// TIA Portal V19 export
FUNCTION_BLOCK "UP_Spuele.GP0x"   // FB1003, LAD
TITLE = Umwälzpumpe Spüle
{ S7_Optimized_Access := 'TRUE' }
// Funktionen:  Entleeren /  Spülen
// stored: AutoNumber false, MemoryReserve 100, SetENOAutomatically false
   VAR RETAIN
      In { ExternalAccessible := 'False'; ExternalVisible := 'False'; ExternalWritable := 'False'} : Struct
         NotHalt : Bool;
         ext_Freigabe : Bool;   // kein Gasalarm, Kein Notstrom
         TW_senkt : Bool;
         Auto : Bool;   // Paneltaste
         Ein : Bool;   // Paneltaste
         FU_betriebsbereit : Bool;
         FU_Stoerung : Bool;
         Niv_TLS : Bool;
         Niv_min : Bool;
         Frg_Niv_CM05 : Bool;
         SRM_Saugseite_auf : Bool;
         SRM_Saugseite_zu : Bool;
         SRM_Druckseite_auf : Bool;
         SRM_Druckseite_zu : Bool;
         GW_p_UP : Bool;
         Betriebsart : USInt := 0;   // Paneltaste
         FU_speed : Int;
         Druck_Pumpe : Real;
      END_STRUCT;
      Param { ExternalAccessible := 'False'; ExternalVisible := 'False'; ExternalWritable := 'False'} : Struct
         SW_Hand : Int;   // [%]
         SW_Auto_AZ : Int;   // [%]
         SW_Auto_aAZ : Int;   // [%]
         Spülzeit : Time;
         DT_Druckaufbau : Time;
         DT_Testzeit : Time;
         SW_Drucktest : Real;
         "Name" : String[12];
      END_STRUCT;
      Zst { ExternalAccessible := 'False'; ExternalVisible := 'False'; ExternalWritable := 'False'} : Struct
         Niveau : USInt;
         Status_GP0x : USInt;
         Status_DT : USInt;
         Restzeit_Spülen : Time;
         Restzeit_DT : Time;
         TON_Spülventil_auf : Bool;
         Spuelen : Bool;
         Spuelen_aktiv : Bool;
         Drucktest_aktiv : Bool;
         Umwaelzen : Bool;
         Zeit_laeuft : Bool;
         Drucktest_ok : Bool;
         Bedienung_erlaubt : Bool;
         speed : Int;   // [%]
      END_STRUCT;
      Mld { ExternalAccessible := 'False'; ExternalVisible := 'False'; ExternalWritable := 'False'} : Struct
         Niv_TLS : Bool;
         Niv_Sensorfehler : Bool;
         GW_p_UP : Bool;
         FU_nicht_bereit : Bool;
         FU_Stoerung : Bool;
         n_Auto : Bool;
         TO_Druckaufbau : Bool;
         Drucktest_ok : Bool;
         DT_Fehler : Bool;
         Pu_Spuelen_Fertig : Bool;
      END_STRUCT;
      Out { ExternalAccessible := 'False'; ExternalVisible := 'False'; ExternalWritable := 'False'} : Struct
         GP0x_Ein : Bool;
         Ventil_Saugseite : Bool;
         Ventil_Druckseite : Bool;
         Spülventil : Bool;
         Ventil_CM05 : Bool;
         Soll_speed : Int;
      END_STRUCT;
   END_VAR
   VAR
      IEC_Timer { ExternalAccessible := 'False'; ExternalVisible := 'False'; ExternalWritable := 'False'} : Struct
         Spülventil_auf { S7_SetPoint := 'True'} : TON_TIME;
         Spülen { S7_SetPoint := 'True'} : TP_TIME;
         GW_p { S7_SetPoint := 'True'} : TON_TIME;
         Drucktest { S7_SetPoint := 'True'} : TP_TIME;
         TO_Druckaufbau { S7_SetPoint := 'True'} : TON_TIME;
         Ventil_CMO5 { S7_SetPoint := 'True'} : TOF_TIME;
      END_STRUCT;
      R_TRIG_Hand_EIN { ExternalAccessible := 'False'; ExternalVisible := 'False'; ExternalWritable := 'False'} : R_TRIG;
   END_VAR
   VAR_TEMP
      Spülzeit : Time;
      Zeit_DT : Time;
      posFl_Hand : Bool;
   END_VAR
   VAR CONSTANT
      Niv_TLS : USInt := 7;
      Niv_Min : USInt := 70;
      Niv_max : USInt := 85;
      Zeit_Ventil_auf : Time := T#1s;
      S1 : USInt := 1;
      S2 : USInt := 2;
      S3 : USInt := 3;
      S4 : USInt := 4;
   END_VAR
BEGIN

REGION Network 1 (SCL): Input
   // Panelbedienung und Sensoren --> Input()
   // Not-Halt
   #In.NotHalt := NOT "DB_PNOZ_IN_Out".In.NH_Frg_Pumpen OR NOT "E_Frg_AbLW";

   // Timer Spülventil AUF
   #IEC_Timer.Spülventil_auf(IN := #Out.Spülventil,
                              PT := #Zeit_Ventil_auf,
                              Q => #Zst.TON_Spülventil_auf);

    // positive Flanke "Hand Ein"
   #R_TRIG_Hand_EIN(CLK := #In.Ein,
                    Q => #posFl_Hand);
END_REGION

REGION Network 2 (SCL): Ansteuerung

   // "Normal"-Betrieb
   #Zst.Bedienung_erlaubt := NOT #In.Ein AND NOT #In.Auto AND NOT #Mld.DT_Fehler;

   //Drucktest rücksetzen
   IF #In.Betriebsart <> 2 OR #Zst.Spuelen_aktiv OR #Zst.Umwaelzen OR NOT #In.Ein THEN
       #Mld.Drucktest_ok := FALSE;
       // #Mld.DT_Fehler := FALSE;
       #Mld.TO_Druckaufbau := FALSE;
       #Zst.Status_DT := 0;
       #Zst.Drucktest_aktiv := FALSE;
   END_IF;
   //Spülmeldung rücksetzen
   IF #In.Betriebsart <> 1 OR NOT #In.Ein THEN
       #Mld.Pu_Spuelen_Fertig := FALSE;
   END_IF;

       CASE #In.Betriebsart OF
           0:  // Umwälzen

               // Spülventil zu
               #Out.Spülventil := FALSE;
               #Out.Ventil_CM05 := FALSE;
               #Zst.Restzeit_Spülen := T#0s;
               // Ventile öffnen
               #Out.Ventil_Saugseite := (#In.Auto OR #In.Ein) AND #In.Niv_TLS AND NOT #In.TW_senkt;
               #Out.Ventil_Druckseite := #Out.Ventil_Saugseite;
               // Wenn geöffnet --> Frg Pumpe
               #Zst.Umwaelzen := #In.SRM_Druckseite_auf AND #In.SRM_Saugseite_auf;
               #Zst.Drucktest_aktiv := FALSE;

           1: // Spülen - nur Hand
               #Zst.Umwaelzen := FALSE;
               #Out.Ventil_Saugseite := FALSE;
               #Out.Ventil_Druckseite := FALSE;

               // Ausschaltverzögert - Druckabbau
               #IEC_Timer.Ventil_CMO5(IN := #Out.Spülventil,
                                      PT := T#3s,
                                      Q => #Out.Ventil_CM05);

                   IF #In.Ein AND #In.Frg_Niv_CM05 THEN
                       IF #posFl_Hand THEN
                           #Zst.Spuelen_aktiv := TRUE;
                       END_IF;

                       #Out.Spülventil := #In.SRM_Druckseite_zu AND #In.SRM_Saugseite_zu AND #Zst.Spuelen_aktiv;

                       #IEC_Timer.Spülen(IN := #Zst.TON_Spülventil_auf,
                                         PT := #Param.Spülzeit,
                                         Q => #Zst.Spuelen,
                                         ET => #Spülzeit);
                       #Zst.Restzeit_Spülen := #Param.Spülzeit - #Spülzeit;

                       IF #Zst.TON_Spülventil_auf AND #In.SRM_Saugseite_zu AND #In.SRM_Druckseite_zu
                           AND NOT #Zst.Spuelen AND #Zst.Spuelen_aktiv THEN
                           #Zst.Spuelen_aktiv := FALSE;
                           #Out.Spülventil := FALSE;
                       END_IF;

                       // Fertig
                       IF NOT #Zst.Spuelen AND NOT #Zst.Spuelen_aktiv AND NOT #Out.Ventil_CM05 THEN
                           #Out.Spülventil := FALSE;
                           #Out.Ventil_CM05 := FALSE;
                           #Zst.Restzeit_Spülen := T#0s;
                           #Mld.Pu_Spuelen_Fertig := TRUE;
                       END_IF;
                   ELSE
                       #Zst.Spuelen := FALSE;
                       #Out.Spülventil := FALSE;
                       #Out.Ventil_CM05 := FALSE;
                       #Zst.Restzeit_Spülen := T#0s;
                   END_IF;

           2: // Spülen + Drucktest - nur Hand
               #Zst.Umwaelzen := FALSE;
               #Out.Ventil_Saugseite := FALSE;
               #Out.Ventil_Druckseite := FALSE;
               IF NOT #Zst.Drucktest_aktiv THEN
                   IF #In.Ein AND #In.Frg_Niv_CM05 THEN
                       IF #posFl_Hand THEN
                           #Zst.Spuelen_aktiv := TRUE;
                       END_IF;

                       #Out.Spülventil := #In.SRM_Druckseite_zu AND #In.SRM_Saugseite_zu AND #Zst.Spuelen_aktiv;
                       #Out.Ventil_CM05 := #Out.Spülventil;

                       #IEC_Timer.Spülen(IN := #Zst.TON_Spülventil_auf,
                                         PT := #Param.Spülzeit,
                                         Q => #Zst.Spuelen,
                                         ET => #Spülzeit);
                       IF #Zst.TON_Spülventil_auf AND #In.SRM_Saugseite_zu AND #In.SRM_Druckseite_zu
                           AND NOT #Zst.Spuelen AND #Zst.Spuelen_aktiv THEN
                           #Zst.Spuelen_aktiv := FALSE;
                       END_IF;
                       #Zst.Restzeit_Spülen := #Param.Spülzeit - #Spülzeit;
                       // Fertig
                       IF NOT #Zst.Spuelen AND NOT #Zst.Spuelen_aktiv THEN
                           #Out.Spülventil := FALSE;
                           #Out.Ventil_CM05 := FALSE;
                           #Zst.Restzeit_Spülen := T#0s;
                           #Zst.Drucktest_aktiv := TRUE;
                           #Zst.Status_DT := #S1;
                       END_IF;
                   ELSE
                       #Zst.Spuelen := FALSE;
                       #Out.Spülventil := FALSE;
                       #Out.Ventil_CM05 := FALSE;
                       #Zst.Restzeit_Spülen := T#0s;
                   END_IF;
               END_IF;

               IF #Zst.Drucktest_aktiv THEN
                   CASE #Zst.Status_DT OF
                       #S1:  //Druckaufbau
                           IF "DB_Temporaer".Drucksensoren_deaktiviert THEN//20.01.22
                               #Zst.Drucktest_ok := TRUE;

                               "Ergebnis_DT"("Name" := #Param.Name,
                                             akt_Zeit := "Uhrzeit".aktDatum,
                                             ok := #Zst.Drucktest_ok,
                                             Fehler := NOT #Zst.Drucktest_ok);

                               #Mld.Drucktest_ok := #Zst.Drucktest_ok;
                               #Mld.DT_Fehler := NOT #Zst.Drucktest_ok;
                               #Zst.Status_DT := #S4;
                           ELSE
                               #Out.Spülventil := #In.SRM_Druckseite_zu AND #In.SRM_Saugseite_zu;
                               #Out.Ventil_CM05 := FALSE;
                               IF (#In.Druck_Pumpe > #Param.SW_Drucktest + 0.25) OR #Mld.TO_Druckaufbau THEN
                                   #Zst.Status_DT := #S2;
                               END_IF;
                               #Zst.Restzeit_DT := #Param.DT_Druckaufbau - #IEC_Timer.TO_Druckaufbau.ET;
                           END_IF;
                       #S2: //Wartezeit
                           #IEC_Timer.Drucktest(IN := NOT #Out.Spülventil,
                                                PT := #Param.DT_Testzeit,
                                                Q => #Zst.Zeit_laeuft,
                                                ET => #Zeit_DT);
                           #Zst.Restzeit_DT := #Param.DT_Testzeit - #Zeit_DT;

                           IF NOT #Zst.Zeit_laeuft AND NOT #Out.Spülventil THEN
                               #Zst.Restzeit_DT := T#0s;
                               #Zst.Status_DT := #S3;
                           END_IF;
                           #Out.Spülventil := FALSE;
                           #Out.Ventil_CM05 := FALSE;
                       #S3:// Überprüfung
                           #Zst.Drucktest_ok := #In.Druck_Pumpe >= #Param.SW_Drucktest;

                           "Ergebnis_DT"("Name" := #Param.Name,
                                         akt_Zeit := "Uhrzeit".aktDatum,
                                         ok := #Zst.Drucktest_ok,
                                         Fehler := NOT #Zst.Drucktest_ok);

                           #Mld.Drucktest_ok := #Zst.Drucktest_ok;
                           #Mld.DT_Fehler := NOT #Zst.Drucktest_ok;
                           #Zst.Status_DT := #S4;
                       #S4: // Ende
                           ;

                   END_CASE;
               END_IF;
       END_CASE;

       // Pumpe an    
       #Out.GP0x_Ein := #Zst.Umwaelzen AND NOT #In.NotHalt AND #In.ext_Freigabe;

       // Geschwindigkeitsvorgabe
       // SEW: 100% == 3000 U/min == 15000 Digits
       IF #Out.GP0x_Ein THEN
           IF #In.Ein THEN
               #Out.Soll_speed := #Param.SW_Hand * 150;
           ELSE
               IF "Uhrzeit".AZ_aktiv THEN
                   #Out.Soll_speed := #Param.SW_Auto_AZ * 150;
               ELSE
                   #Out.Soll_speed := #Param.SW_Auto_aAZ * 150;
               END_IF;
           END_IF;
       ELSE
           #Out.Soll_speed := 0;
       END_IF;
END_REGION

REGION Network 3 (SCL): Überwachung / Meldungen
   // Trockenlaufschutz
   #Mld.Niv_TLS := NOT #In.Niv_TLS;

   // Zeitüberschreitung Druckaufbau
   #IEC_Timer.TO_Druckaufbau(IN := #Zst.Status_DT = #S1,
                             PT := #Param.DT_Druckaufbau,
                             Q => #Mld.TO_Druckaufbau);

   // Grenzwert Druck
   #IEC_Timer.GW_p(IN :=#Out.GP0x_Ein AND #In.GW_p_UP,
                   PT := T#3s,
                   Q => #Mld.GW_p_UP);
   // Frequenzumrichter 24V-Betrieb
   #Mld.FU_nicht_bereit := NOT #In.FU_betriebsbereit AND NOT #In.NotHalt;
   // Störung Frequenzumrichter
   #Mld.FU_Stoerung := #In.FU_Stoerung AND NOT #In.NotHalt;
   // nicht in Automatik
   #Mld.n_Auto := FALSE; //NOT #In.Auto AND "DB_ANLAGE".BA.Automat_ein;
END_REGION

REGION Network 4 (SCL): --> Visu
   // Status Pumpe
   "Status_E0A"(Hand := #In.Ein,
                Auto := #In.Auto,
                SonderModus_PumpeSpuelen:=#Zst.Spuelen,
                Stoerung := #In.FU_Stoerung OR NOT #In.FU_betriebsbereit,
                Ausgang := #Out.GP0x_Ein,
                StatusByte => #Zst.Status_GP0x);

   // Ist-Geschwindigkeit FU
   // SEW: 100% == 3000 U/min == 15000 Digits
   #Zst.speed := #In.FU_speed / 150; // in[%]

   // Anzeige Füllstand
   "Niv_Visu"(Niv_1 := #In.Niv_TLS,
              Niv_2 := #In.Niv_min,
              Niv_3 := FALSE,
              Niv_4 := FALSE,
              Niv_5 := FALSE,
              Niv_6 := FALSE,
              Wert_1 := #Niv_TLS,
              Wert_2 := #Niv_max,
              Wert_3 := 0,
              Wert_4 := 0,
              Wert_5 := 0,
              Wert_6 := 0,
              Niveau => #Zst.Niveau,
              Niv_Err => #Mld.Niv_Sensorfehler);
END_REGION
END_FUNCTION_BLOCK
